//LED state of the safety controller PNOZmulti 2
TYPE ST_LEDState :
STRUCT
    nLEDState: USINT;
END_STRUCT
END_TYPE

(* stored: Version 1.1.0.1
   DUT ST_LEDState: Id {f261f142-fde3-0208-2395-07dc6293304d} *)
